Xinje XDPPro project, PLC1: XL5E-16 (software 3.7.14b 2022-06-24)

PROGRAM 梯形图

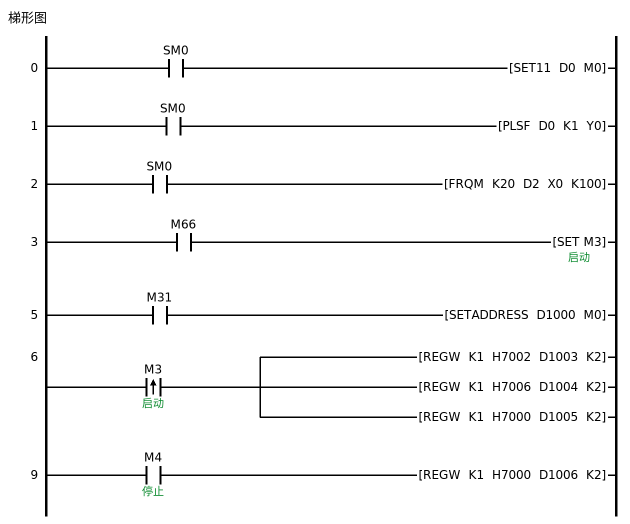
LD     SM0
SET11  D0 M0
LD     SM0
PLSF   D0 K1 Y0
LD     SM0
FRQM   K20 D2 X0 K100
LD     M66
SET    M3	; 启动
LD     M31
SETADDRESS D1000 M0
LDP    M3	; 启动
REGW   K1 H7002 D1003 K2
REGW   K1 H7006 D1004 K2
REGW   K1 H7000 D1005 K2
LD     M4	; 停止
REGW   K1 H7000 D1006 K2

C FUNCTION BLOCK set11.fcb
/* #EXPORT_ENTRY_BEGIN(SET11)
//    类型              模式             个数               映射          注释
W = { type = "PINT16S", mode = [In,Out], count = "unknown", map = [D,HD], comment = "" }
B = { type = "BIT"    , mode = [In,Out], count = "unknown", map = [M,HM], comment = "" }
#EXPORT_ENTRY_END */
/*************************************************************************
 * FunctionBlockName:  SET11
 * Version:            1.0.0
 * Author:             
 * UpdateTime:         2022-10-10 10:25:17
 * Comment:            
**************************************************************************/

/**
 * @summary 
 * @param W 
 * @param B 
 */
void SET11(PINT16S W,BIT B)
{
	#define SysRegAddr_HD_D_HM_M
    D[0] = 60000;
}

C FUNCTION BLOCK setaddress.fcb
/* #EXPORT_ENTRY_BEGIN(SETADDRESS)
//    类型              模式             个数               映射          注释
W = { type = "PINT16S", mode = [In,Out], count = "unknown", map = [D,HD], comment = "" }
B = { type = "BIT"    , mode = [In,Out], count = "unknown", map = [M,HM], comment = "" }
#EXPORT_ENTRY_END */
/*************************************************************************
 * FunctionBlockName:  SETADDRESS
 * Version:            1.0.0
 * Author:             
 * UpdateTime:         2022-10-10 16:33:40
 * Comment:            
**************************************************************************/

/**
 * @summary 
 * @param W 
 * @param B 
 */
void SETADDRESS(PINT16S W,BIT B)
{
	#define SysRegAddr_HD_D_HM_M
   D[1000] = 0x7002;
   D[1001]  = 0x7006;
   D[1002]  = 0x7000;
   D[1003] = 1000;
   D[1004] = 1500;
   D[1005]  = 1;
   D[1006] = 6;
    return;
}